// TIA Portal project "P3" (V17)

(* hardware
DEVICE "S7-1500/ET200MP station_1"  S7-1500 station
   slot 0: "Rail_0"  Rack  6ES7 590-1***0-0AA0
   slot 1: "PLC_1"  CPU 1515-2 PN  6ES7 515-2AM02-0AB0  V2.9
      slot 3: "CPU display_1"  6ES7591-1BA00-0AA0
      slot 32768: "PROFINET interface_1"  X1
         slot 32769: "Port_1"  X1 P1
         slot 32770: "Port_2"  X1 P2
      slot 33024: "PROFINET interface_2"  X2
         slot 33025: "Port_1"  X2 P1
      slot 34817: "Virtual CP interface port_1"  Virtual CP interface port  Virtual CP interface port
*)

// ===== PLC "PLC_1"  CPU 1515-2 PN =====

VAR_GLOBAL   // PLC tag table "Default tag table"
   "START PB" AT %E0.0 : Bool;
   "STOP PB" AT %E0.1 : Bool;
   "YELLOW SELECTION" AT %E0.2 : Bool;
   "BLUE SELECTION" AT %E0.3 : Bool;
   "GREEN SELECTION" AT %E0.4 : Bool;
   "SWITCH ON/OFF" AT %M2.0 : Bool;
   "CYCLE ON" AT %A0.0 : Bool;
   "YELLOW CONTROL VALVULE" AT %A0.1 : Bool;
   "BLUE CONTROL VALVULE" AT %A0.2 : Bool;
END_VAR

ORGANIZATION_BLOCK "Main"   // OB1, LAD, ProgramCycle
TITLE = "Main Program Sweep (Cycle)"
{ S7_Optimized_Access := 'TRUE' }
VERSION : 0.1
   VAR_INPUT
      Initial_Call : Bool;   // Initial call of this OB
      Remanence : Bool;   // =True, if remanent data are available
   END_VAR
BEGIN

REGION Network 1: CYCLE ON
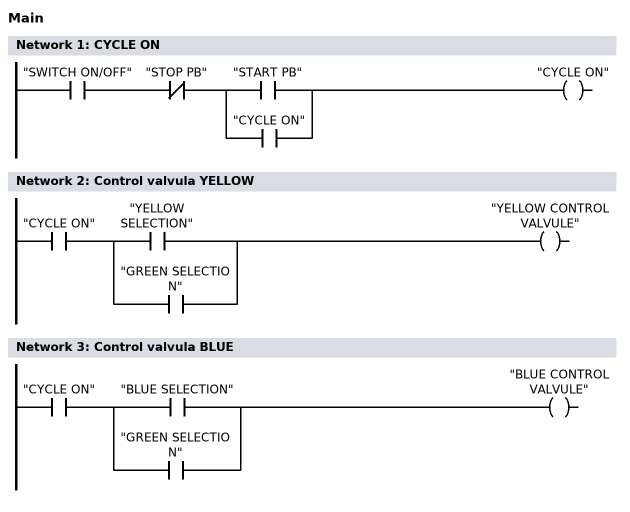
   RUNG wire#powerrail
      Contact( "SWITCH ON/OFF" )
      I_Contact( "STOP PB" )
      wire#w1
      Contact( "START PB" )
      wire#w2
      Coil( "CYCLE ON" )
   END_RUNG
   RUNG wire#w1
      Contact( "CYCLE ON" )
   END_RUNG wire#w2
   // the same network as SCL:
   "CYCLE ON" := "SWITCH ON/OFF" AND NOT "STOP PB" AND ("START PB" OR "CYCLE ON");
END_REGION

REGION Network 2: Control valvula YELLOW
   RUNG wire#powerrail
      Contact( "CYCLE ON" )
      wire#w1
      Contact( "YELLOW SELECTION" )
      wire#w2
      Coil( "YELLOW CONTROL VALVULE" )
   END_RUNG
   RUNG wire#w1
      Contact( "GREEN SELECTION" )
   END_RUNG wire#w2
   // the same network as SCL:
   "YELLOW CONTROL VALVULE" := "CYCLE ON" AND ("YELLOW SELECTION" OR "GREEN SELECTION");
END_REGION

REGION Network 3: Control valvula BLUE
   RUNG wire#powerrail
      Contact( "CYCLE ON" )
      wire#w1
      Contact( "BLUE SELECTION" )
      wire#w2
      Coil( "BLUE CONTROL VALVULE" )
   END_RUNG
   RUNG wire#w1
      Contact( "GREEN SELECTION" )
   END_RUNG wire#w2
   // the same network as SCL:
   "BLUE CONTROL VALVULE" := "CYCLE ON" AND ("BLUE SELECTION" OR "GREEN SELECTION");
END_REGION
END_ORGANIZATION_BLOCK